PROGRAM MAIN
VAR




state : MS;

NewTable 	: FB_NewTable;
WriteDB		: FB_DB_Write;



// current file time

		fbSystemTime    : GETSYSTEMTIME;
        timeAsFileTime  : T_FILETIME;
        timeAsDT        : DT;
// Measurement trigger
		trig			: BOOL;

		
// Run Python script for measurement stuff
		runpython		: BOOL:=TRUE;
		Start_py_script : NT_StartProcess;
		
// Run Blockly & FRANKA Desk

//        bStartscript 	: BOOL := TRUE;
        bBusy 			: BOOL := FALSE;
        Start_py_script1 : NT_StartProcess;
		
// IPC Shut Down
		shutdown	:shutdown; 
	
// LED confirmation counter
k: INT :=1;

// Blink Funktion
fbBlinker_grun		:	FB_Blinker;	
fbBlinker_rot		:	FB_Blinker;
fbBlinker_weis		:	FB_Blinker;
green_init			:	BOOL;

// Init_delay
   Delay_startup		: TON;
   Delay			: TON;
   Start_init		: BOOL:=FALSE;
   Delay_init		: BOOL;
   
	clear: INT;
END_VAR

fbSystemTime( timeLoDW =>timeAsFileTime.dwLowDateTime , timeHiDW =>timeAsFileTime.dwHighDateTime );
timeAsDT := FILETIME_TO_DT( timeAsFileTime );

GVL_IO.FRANKA_Marker0 				REF= GVL.mb_Output_Coils[0];
GVL_IO.FRANKA_home1	 				REF= GVL.mb_Output_Coils[1];
GVL_IO.PCB_Marker2	 				REF= GVL.mb_Output_Coils[2];
GVL_IO.FRANKA_MPoint_reached3		REF= GVL.mb_Output_Coils[3];
GVL_IO.FRANKA_Measurement_finished4	REF= GVL.mb_Output_Coils[4];
GVL_IO.FRANKA_PCB_Picked5			REF= GVL.mb_Output_Coils[5];
GVL_IO.FRANKA_PCB_Placed6			REF= GVL.mb_Output_Coils[6];
GVL_IO.FRANKA_ready_to_start		REF= GVL.mb_Output_Coils[7];
GVL_IO.PLC_Measure_Finished0		REF= GVL.mb_Input_Coils[0];
GVL_IO.PLC_confirm_PCB_placement1	REF= GVL.mb_Input_Coils[1];
GVL_IO.PLC_Start_trigger			REF= GVL.mb_Input_Coils[2];

shutdown(Trig:=GVL.Grau_Schalter);
IF GVL.Stop_Schalter=TRUE THEN
	state:=MS.Reset;
END_IF


GVL.Data.PCB_Batch_ID:= GVL_Persistent.PCB_Batch_ID;




CASE state OF


MS.Reset : 	
			// Reset HMI
				IF clear<9 THEN
					GVL.Visu_Data[clear].PCB_Batch_ID:=0;
					GVL.Visu_Data[clear].PCB_ID:=0;
					GVL.Visu_Data[clear].PCB_no_defects:='';
					GVL.Visu_Data[clear].Measure1InTol:='';
					GVL.Visu_Data[clear].Measure2InTol:='';
					GVL.Visu_Data[clear].Measure3InTol:='';
					GVL.PLC_Data[clear].MeasureInTol[1]:='';
					GVL.PLC_Data[clear].MeasureInTol[2]:='';
					GVL.PLC_Data[clear].MeasureInTol[3]:='';					
					clear:=clear+1;
				END_IF

			
			// LEDs off
				GVL.LED1:=FALSE;
				GVL.LED2:=FALSE;
				GVL.LED3:=FALSE;
				GVL.LED4:=FALSE;
				GVL.LED5:=FALSE;
				GVL.LED6:=FALSE;
				GVL.LED7:=FALSE;
				GVL.LED8:=FALSE;
			//
            fbBlinker_weis(bStart:=TRUE , tPeriode:= T#1S, bBlinker=>GVL.Schalterlichtweis);
			GVL.Schalterlichtgrun:=FALSE;
			GVL.bStartBlockly := FALSE;
			GVL.measure_n:=1;
			GVL.pcb_n:=1;
			Start_init:=FALSE;
			GVL_IO.FRANKA_ready_to_start:=FALSE;
			Delay(IN:=FALSE);
			IF GVL.Grau_Schalter=TRUE THEN
				state:= MS.Start;
				// Batch ID Increment
				GVL_Persistent.PCB_Batch_ID:=GVL_Persistent.PCB_Batch_ID+1;
			END_IF
			
MS.Init_delay:
				Delay_startup(IN:=TRUE, PT:= T#10S, Q=>Start_init, ET=>);
				IF Start_init=TRUE THEN
					Start_init:=FALSE;
					state:=MS.Initialization;
				END_IF

MS.Initialization:

			// LEDs off
				GVL.LED1:=FALSE;
				GVL.LED2:=FALSE;
				GVL.LED3:=FALSE;
				GVL.LED4:=FALSE;
				GVL.LED5:=FALSE;
				GVL.LED6:=FALSE;
				GVL.LED7:=FALSE;
				GVL.LED8:=FALSE;
				

				GVL.Schalterlichtweis:=TRUE;
				GVL.schalterspannung:= TRUE;
			// Initialize Blockly & FRANKA Desk
					
			    IF GVL.bStartBlockly = TRUE AND bBusy = FALSE THEN
        			Start_py_script1(
            		NETID := '',
            		PATHSTR := 'blocklenium',
            		DIRNAME := 'C:\Users\Administrator\Desktop',
     				COMNDLINE := '--insecure-con --login-required -b PCB_Measure.url -u http://192.168.2.2/desk/',
					//COMNDLINE := '--insecure-con --login-required -b PCB_Handling.url -u http://192.168.2.2/desk/',
                	START := TRUE,
            		BUSY => bBusy
        			);
       			 	GVL.bStartBlockly := FALSE;
					//bBusy:= FALSE;
    			END_IF
			
				
				
		// Initialize Measurement script
		
			IF runpython = TRUE THEN	
				Start_py_script(NETID:='',
				PATHSTR:= 'bkpads',
				DIRNAME:= 'C:\Users\Administrator\Desktop\',
				COMNDLINE:='-c COM4',
				Start:=TRUE,
				TMOUT:=T#1S);
				runpython:=FALSE;
			 END_IF		
		

//			IF runpython = TRUE THEN	
//				Start_py_script(NETID:='',
//				PATHSTR:= 'C:\Python38\python.exe',
//				DIRNAME:= 'C:\Users\Administrator\Desktop\',
//				COMNDLINE:='C:\Users\Administrator\Desktop\bkpads.py',
//				Start:=TRUE,
//				TMOUT:=T#1S);
//				runpython:=FALSE;
//			 END_IF
			
			// Initializes, settings for measurement
			GVL.pcb_n:=1;
			GVL.pcb_max:=8;
			GVL.measure_n:=1;
			GVL.measure_max:=3;
			Initialize_Measurement_Values(); // Set Measurement references, tolerances & Types for measurement points on PCB
			
			IF GVL.Measurement_Init=TRUE THEN
			Delay_init:=TRUE;
			// Batch ID Increment
			GVL_Persistent.PCB_Batch_ID:=GVL_Persistent.PCB_Batch_ID+1;
			state:=MS.Start;
			;
			END_IF
			
			// Initialize table
			GVL.ActiveTable:='PCB_Test_Results';
			NewTable ();

MS.Restart:

			//
			GVL.Schalterlichtgrun:=FALSE;
			GVL.bStartBlockly := FALSE;
			GVL.measure_n:=1;
			GVL.pcb_n:=1;
			Start_init:=FALSE;
			Delay(IN:=FALSE);
			fbBlinker_grun(bStart:=Start_init , tPeriode:= T#1S, bBlinker=>GVL.Schalterlichtgrun);
			IF GVL.Start_Schalter= TRUE THEN			
				GVL.LED1:=FALSE;
				GVL.LED2:=FALSE;
				GVL.LED3:=FALSE;
				GVL.LED4:=FALSE;
				GVL.LED5:=FALSE;
				GVL.LED6:=FALSE;
				GVL.LED7:=FALSE;
				GVL.LED8:=FALSE;
				state:=MS.Start;		
			END_IF
					
			
			
			
			
			
MS.Start :	
			clear:=1;
			GVL.bStartBlockly := TRUE;
			Delay(IN:=Delay_init, PT:= T#30S, Q=>Start_init);
			
			IF Start_init = TRUE AND GVL_IO.FRANKA_ready_to_start=FALSE THEN
				state:= MS.FRANKA_ERROR;
			END_IF
			
		    fbBlinker_grun(bStart:=Start_init , tPeriode:= T#1S, bBlinker=>GVL.Schalterlichtgrun);
			
			
			GVL.Schalterlichtrot:=TRUE;
			IF GVL.Start_Schalter= TRUE THEN
				GVL_IO.PLC_Start_trigger:= TRUE;
			END_IF
			
			
			IF GVL_IO.FRANKA_Marker0 = TRUE THEN 
				GVL.Schalterlichtweis:= FALSE;
				GVL_IO.PLC_Start_trigger:= FALSE;
				fbBlinker_grun(bStart:=FALSE);
				state:=MS.FRANKA_Pick_and_place_PCB;
			ELSE ;
			END_IF
					
				
MS.FRANKA_Pick_and_place_PCB:

				IF GVL.pcb_n<=GVL.pcb_max THEN
					IF GVL_IO.FRANKA_PCB_Picked5 = TRUE THEN
						GVL_IO.PLC_confirm_PCB_placement1:=FALSE;
						state:=MS.FRANKA_Measure;
					END_IF
					ELSE;
						// finish program and write report from database
						state:=MS.Restart;
				END_IF
				
MS.FRANKA_Measure: 			
				IF GVL_IO.FRANKA_Measurement_finished4 = FALSE AND GVL_IO.FRANKA_MPoint_reached3 = TRUE THEN					
						GVL.sMeas_type:=GVL.PLC_Data[GVL.pcb_n].Measure_Type[GVL.measure_n];	// set type  
						IF  trig=FALSE THEN
							GVL.bMeas_start:= TRUE; // Trigger Measurement
							GVL_IO.PLC_Measure_Finished0:= FALSE;
							trig:=TRUE;
						END_IF
						IF GVL.bMeas_ready =TRUE THEN
							GVL.PLC_Data[GVL.pcb_n].Measure_Result[GVL.measure_n]:=GVL.rMeas_01;
							//rMeas_02	: 	REAL;	// Measurement result 2
							IF GVL.PLC_Data[GVL.pcb_n].Measure_Result[GVL.measure_n]<(GVL.PLC_Data[GVL.pcb_n].Measure_Reference[GVL.measure_n]+GVL.PLC_Data[GVL.pcb_n].Measure_Tolerance[GVL.measure_n]) AND GVL.PLC_Data[GVL.pcb_n].Measure_Result[GVL.measure_n]>(GVL.PLC_Data[GVL.pcb_n].Measure_Reference[GVL.measure_n]-GVL.PLC_Data[GVL.pcb_n].Measure_Tolerance[GVL.measure_n]) THEN
								GVL.PLC_Data[GVL.pcb_n].MeasureInTol[GVL.measure_n]:= 'Yes';

								ELSE
								GVL.PLC_Data[GVL.pcb_n].MeasureInTol[GVL.measure_n]:= 'No'; // test LED's YES otherwise No
								GVL.PLC_Data[GVL.pcb_n].PCB_no_defects:= 'defect';
								GVL.Visu_Data[GVL.pcb_n].PCB_no_defects:='defect';
							END_IF
							
							GVL_IO.PLC_Measure_Finished0:= TRUE;							
							IF GVL_IO.FRANKA_Marker0 =TRUE THEN
								state:=MS.DB_Write;
							END_IF
						END_IF
				END_IF

		
MS.DB_Write:
		// Visu Data
		GVL.Visu_Data[GVL.pcb_n].PCB_Batch_ID:=GVL_Persistent.PCB_Batch_ID;
		GVL.Visu_Data[GVL.pcb_n].PCB_ID:=GVL.pcb_n;
		GVL.Visu_Data[GVL.pcb_n].Measure1InTol:=GVL.PLC_Data[GVL.pcb_n].MeasureInTol[1];
		GVL.Visu_Data[GVL.pcb_n].Measure2InTol:=GVL.PLC_Data[GVL.pcb_n].MeasureInTol[2];
		GVL.Visu_Data[GVL.pcb_n].Measure3InTol:=GVL.PLC_Data[GVL.pcb_n].MeasureInTol[3];
		

		GVL.Data.PCB_ID:=GVL.pcb_n;
		GVL.Data.Measurement_ID:=GVL.measure_n;
		GVL.Data.Measure_Type:=GVL.PLC_Data[GVL.pcb_n].Measure_Type[GVL.measure_n];
		GVL.Data.TimeStamp:= timeASDT;
		GVL.Data.FreeFromDefects:=GVL.PLC_Data[GVL.pcb_n].MeasureInTol[GVL.measure_n];
		GVL.Data.Measure_Type:= GVL.PLC_Data[GVL.pcb_n].Measure_Type[GVL.measure_n];
		GVL.Data.Measure_Result:= GVL.PLC_Data[GVL.pcb_n].Measure_Result[GVL.measure_n];
		GVL.Data.Measure_Reference:= GVL.PLC_Data[GVL.pcb_n].Measure_Reference[GVL.measure_n];
		GVL.Data.Measure_Tolerance:= GVL.PLC_Data[GVL.pcb_n].Measure_Tolerance[GVL.measure_n];
		WriteDB ();
		IF GVL.Writing_finished=TRUE THEN
			GVL.write_state:=0;
			GVL_IO.FRANKA_MPoint_reached3:=FALSE;
			GVL.measure_n:=GVL.measure_n+1;
			trig:=FALSE;
			GVL.bMeas_ready:=FALSE;
		END_IF
																
		IF GVL.measure_n=GVL.measure_max+1 AND GVL.Writing_finished=TRUE THEN
			GVL_IO.PLC_Measure_Finished0:= FALSE;
			GVL.measure_n:=1;
			state:=MS.FRANKA_Place_PCB;	
			ELSE
			state:=MS.FRANKA_Measure;
		END_IF

				
							
MS.FRANKA_Place_PCB:
				
						IF GVL_IO.FRANKA_PCB_Placed6 = TRUE THEN
							
							GVL_IO.PLC_confirm_PCB_placement1:=TRUE;
							state:=MS.LED_confirmation;
							GVL_IO.FRANKA_PCB_Placed6:= FALSE;
						END_IF

MS.LED_confirmation:			
				// No defects in PCB?
				IF k<=GVL.measure_max THEN
					IF GVL.PLC_Data[GVL.pcb_n].MeasureInTol[k]='No' THEN
						GVL.pcb_n:=GVL.pcb_n+1;
						k:=1;
						state:=MS.FRANKA_Pick_and_place_PCB;			
					ELSE
						IF k=GVL.measure_max AND GVL.PLC_Data[GVL.pcb_n].MeasureInTol[k]='No' THEN
							GVL.pcb_n:=GVL.pcb_n+1;
							state:=MS.FRANKA_Pick_and_place_PCB;
							ELSE
							k:=k+1;
						END_IF
					END_IF
				ELSE
					CASE GVL.pcb_n OF
						1: GVL.LED1:=TRUE;
						   GVL.Visu_Data[1].PCB_no_defects:='Yes';
						2: GVL.LED2:=TRUE;
						   GVL.Visu_Data[2].PCB_no_defects:='Yes';
						3: GVL.LED3:=TRUE;
						   GVL.Visu_Data[3].PCB_no_defects:='Yes';
						4: GVL.LED4:=TRUE;
						   GVL.Visu_Data[4].PCB_no_defects:='Yes';
						5: GVL.LED5:=TRUE;
						   GVL.Visu_Data[5].PCB_no_defects:='Yes';
						6: GVL.LED6:=TRUE;
						   GVL.Visu_Data[6].PCB_no_defects:='Yes';
						7: GVL.LED7:=TRUE;
						   GVL.Visu_Data[7].PCB_no_defects:='Yes';
						8: GVL.LED8:=TRUE;
						   GVL.Visu_Data[8].PCB_no_defects:='Yes';
					END_CASE
						GVL.pcb_n:=GVL.pcb_n+1;
						k:=1;
						state:=MS.FRANKA_Pick_and_place_PCB;	
				END_IF	

	
MS.FRANKA_ERROR:
fbBlinker_rot(bStart:=TRUE , tPeriode:= T#0.2S, bBlinker=>GVL.Schalterlichtrot);
fbBlinker_grun(bStart:=TRUE , tPeriode:= T#1S, bBlinker=>GVL.Schalterlichtgrun);
fbBlinker_weis(bStart:=TRUE , tPeriode:= T#1S, bBlinker=>GVL.Schalterlichtweis);

MS.measurebackup:
				IF GVL_IO.FRANKA_Measurement_finished4 = FALSE AND GVL_IO.FRANKA_MPoint_reached3 = TRUE THEN					
						GVL.sMeas_type:=GVL.PLC_Data[GVL.pcb_n].Measure_Type[GVL.measure_n];	// set type  
						IF  trig=FALSE THEN
							GVL.bMeas_start:= TRUE; // Trigger Measurement
							GVL_IO.PLC_Measure_Finished0:= FALSE;
							trig:=TRUE;
						END_IF
						IF GVL.bMeas_ready =TRUE THEN
							GVL.PLC_Data[GVL.pcb_n].Measure_Result[GVL.measure_n]:=GVL.rMeas_01;
							//rMeas_02	: 	REAL;	// Measurement result 2
							IF GVL.PLC_Data[GVL.pcb_n].Measure_Result[GVL.measure_n]<(GVL.PLC_Data[GVL.pcb_n].Measure_Reference[GVL.measure_n]+GVL.PLC_Data[GVL.pcb_n].Measure_Tolerance[GVL.measure_n]) AND GVL.PLC_Data[GVL.pcb_n].Measure_Result[GVL.measure_n]>(GVL.PLC_Data[GVL.pcb_n].Measure_Reference[GVL.measure_n]-GVL.PLC_Data[GVL.pcb_n].Measure_Tolerance[GVL.measure_n]) THEN
								GVL.PLC_Data[GVL.pcb_n].MeasureInTol[GVL.measure_n]:= 'Yes';

								ELSE
								GVL.PLC_Data[GVL.pcb_n].MeasureInTol[GVL.measure_n]:= 'No'; // test LED's YES otherwise No
								GVL.PLC_Data[GVL.pcb_n].PCB_no_defects:= 'defect';
							END_IF
							
							GVL_IO.PLC_Measure_Finished0:= TRUE;
							
							
							IF GVL_IO.FRANKA_Marker0 =TRUE THEN
								GVL_IO.FRANKA_MPoint_reached3:=FALSE;
								GVL.measure_n:=GVL.measure_n+1;
								trig:=FALSE;
								GVL.bMeas_ready:=FALSE;
								
								
								IF GVL.measure_n=GVL.measure_max+1 THEN
									GVL_IO.PLC_Measure_Finished0:= FALSE;
									GVL.measure_n:=1;
									//state:=MS.FRANKA_Place_PCB;
									state:=MS.FRANKA_Place_PCB;	
								END_IF
							END_IF
						END_IF
				END_IF


				
				
//DB Write Backup
				GVL.Data.PCB_ID:=GVL.pcb_n;
				GVL.Data.Measurement_ID:=GVL.measure_n;
				GVL.Data.Measure_Type:=GVL.PLC_Data[GVL.pcb_n].Measure_Type[GVL.measure_n];
				GVL.Data.TimeStamp:= timeASDT;
				GVL.Data.FreeFromDefects:='Yes';
				GVL.Data.Measure_Type:= 'Resistance';
				GVL.Data.Measure_Result:= 43.3;
				GVL.Data.Measure_Reference:= 4.4;
				GVL.Data.Measure_Tolerance:= 0.2;
				WriteDB ();
				IF GVL.Writing_finished=TRUE THEN
				GVL.write_state:=0;
				END_IF

END_CASE

END_PROGRAM

(* stored: Version 1.1.0.1, ProductVersion 3.1.4024.3
   POU MAIN: Id {2a30b9d8-1355-45f8-afa5-d9af0254be3a}, SpecialFunc None *)
